# EPICS substitutions: viocs/bo_ps/bo_psApp/Db/family.substitutions
file "db/family.db" {
    pattern { family }

        { "QD-FAM" }
        { "QF-FAM" }
        { "SD-FAM" }
        { "SF-FAM" }
        { "BEND-FAM-A" }
        { "BEND-FAM-B" }
}
